# EPICS autosave request: iocBoot/ioc1/dbSave/auto_settings.req
file BP_Kb_.req  P=23d:
file BP_Mo_.req  P=23d:
file CS_Ah_.req  P=23d:
file CS_Av_.req  P=23d:
file KB_Hy_.req  P=23d:
file KB_Hz_.req  P=23d:
file KB_Vy_.req  P=23d:
file KB_Vz_.req  P=23d:
file MO_En_.req  P=23d:
file MO_Ps_.req  P=23d:
file MO_Tn1_.req P=23d:
file MO_Tn2_.req P=23d:
file WS_Ah_.req  P=23d:
file WS_Av_.req  P=23d:

% file CCD_Lp_.req P=23d:
% file CCD_St_.req P=23d:
% file GO_Om_.req  P=23d:
% file GO_Kp_.req  P=23d:
% file GO_Cr_.req  P=23d:
% file GO_St_.req  P=23d:
% file FLU_Di_.req P=23d:
% file BD_Dh_.req  P=23d:
% file BD_Dv_.req  P=23d:
% file GS_St_.req  P=23d:
% file GS_Av_.req  P=23d:
% file GS_Ah_.req  P=23d:
% file BS_Ps_.req  P=23d:
% file TV_V1_.req  P=23d:
% file TV_V2_.req  P=23d:
% file SH_Ps_.req  P=23d:

file COL_St_.req  P=23d:
% file XY_P1_.req  P=23d:
% file XY_P2_.req  P=23d:
% file XY_P3_.req  P=23d:
% file XY_P4_.req  P=23d:
% file XY_P5_.req  P=23d:
% file XY_P6_.req  P=23d:
% file XY_P7_.req  P=23d:
% file XY_P8_.req  P=23d:
% file XY_P9_.req  P=23d:
% %%% file XY_P10_.req P=23d:
% %%% file XY_P11_.req P=23d:
% file XY_P12_.req P=23d:
% file XY_P13_.req P=23d:
% file XY_P14_.req P=23d:
% file XY_P15_.req P=23d:
% file XY_P16_.req P=23d:
% file HS_Ah_.req  P=23d:
% file HS_Av_.req  P=23d:
